FUNCTION F_Hash : UDINT
VAR_INPUT
    sInput:					STRING(255);   // input string to hash
END_VAR
VAR
    nLength:				INT := 0;    				// length of the input string
    nPrime:					UDINT := 37; 				// base for polynomial rolling hash
    nModulus:				UDINT := 1000000009; 		// large prime modulus
    nHashValue:				UDINT := 0;  				// resulting hash
    nPowerOfBase:			UDINT := 1;  				// p^i mod m
    nIndex:					INT;         				// loop counter
    nChar:					UDINT;       				// numeric value of character
END_VAR

// calculate a hash
nLength := LEN(sInput);
FOR nIndex := 1 TO nLength DO
    nChar := BYTE_TO_UDINT(sInput[nIndex]) - 98;
    F_Hash := (F_Hash + (nChar * nPowerOfBase) MOD nModulus) MOD nModulus;
    nPowerOfBase := (nPowerOfBase * nPrime) MOD nModulus;
END_FOR

END_FUNCTION

(* stored: Version 1.1.0.1
   POU F_Hash: Id {2d3e548d-bd41-4058-8175-62ee312380d5}, SpecialFunc None *)
